Staubli VAL3: IsInput.pgx

program IsInput(num x_nIOid (dimensions=1), bool& x_bRes (dimensions=1))
begin

  x_bRes=false
  switch true

    //序号为0
    //    case x_nIOid==0
    //      x_bRes=true
    //    break

    //数字量输入
    case x_nIOid>0 and x_nIOid<67
      x_bRes=true
    break


    //数字量输出
    case x_nIOid>134 and x_nIOid<=140
      x_bRes=false
    break

    //数字量输入
    case x_nIOid>140 and x_nIOid<=144
      x_bRes=true
    break

    //数字量输出
    case x_nIOid>144 and x_nIOid<=164
      x_bRes=false
    break

    //延时等待
    case x_nIOid==165
      x_bRes=true
    break


    //收弧时间
    case x_nIOid==166
      x_bRes=true
    break


    //收弧长度
    case x_nIOid==167
      x_bRes=false
    break


    default
    break
  endSwitch

end
